SUBAPPLICATION RedWhiteBackground2C (* Hintergrundfarbe (TRUE -> Rot, FALSE -> Weiß) für 2 Objekte (Kompakt) *)
  (* Standard: 61499-2 *)
  (* Version 1.0, 2023-02-06, franz, Meisterschulen am Ostbahnhof *)
  PACKAGE MyLib::sys;
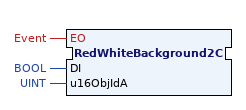
  EVENT_INPUT
    EO;
  END_EVENT
  VAR_INPUT
    DI : BOOL;
    u16ObjIdA : UINT;
  END_VAR
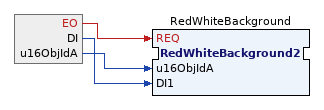
  SUBAPPS
    RedWhiteBackground : MyLib::sys::RedWhiteBackground2;
  END_SUBAPPS
  EVENT_CONNECTIONS
    EO TO RedWhiteBackground.REQ;
  END_CONNECTIONS
  DATA_CONNECTIONS
    u16ObjIdA TO RedWhiteBackground.u16ObjIdA;
    DI TO RedWhiteBackground.DI1;
  END_CONNECTIONS
END_SUBAPPLICATION
